// TIA Portal V18 export
TagTable "Screen1_HMI_Tags"
  CV3201_Nuoc_Bon1_M : Real  (PLC tag CV3201_Nuoc_Bon1_M, HMI_Connection_1, 1 s)   // Col1 Bon1, hang CV, PLC_1 addr=%MD1200
  CV3206_Hoi_Bon2_M : Real  (PLC tag CV3206_Hoi_Bon2_M, HMI_Connection_1, 1 s)   // Col2 Bon2, hang CV, PLC_1 addr=%MD1208
  CV3211_Nuoc_Bon3_M : Real  (PLC tag CV3211_Nuoc_Bon3_M, HMI_Connection_2, 1 s)   // Col4 Bon3, hang CV, PLC_2 addr=%MD1216 - BLOCKER
  CV3216_Hoi_Bon4_M : Real  (PLC tag CV3216_Hoi_Bon4_M, HMI_Connection_2, 1 s)   // Col3 Bon4, hang CV, PLC_2 addr=%MD1224 - BLOCKER
  CV3304_Nuoc_Lam_Mat_M : Real  (PLC tag CV3304_Nuoc_Lam_Mat_M, HMI_Connection_1, 1 s)   // x=832,y=741, CV nuoc lam mat, PLC_1 addr=%MD1232, format=999.9 (%)
  FQ3200_Bon1_Eff : Real  (PLC tag FQ3200_Bon1_Eff, HMI_Connection_1, 1 s)   // Col1 Bon1, hang FQ, PLC_1 addr=%MD712
  FQ3205_Bon2_Eff : Real  (PLC tag FQ3205_Bon2_Eff, HMI_Connection_1, 1 s)   // Col2 Bon2, hang FQ, PLC_1 addr=%MD744
  FQ3210_Bon3_Eff : Real  (PLC tag FQ3210_Bon3_Eff, HMI_Connection_2, 1 s)   // Col4 Bon3, hang FQ, PLC_2 addr=%MD776 - BLOCKER
  FQ3215_Bon4_Eff : Real  (PLC tag FQ3215_Bon4_Eff, HMI_Connection_2, 1 s)   // Col3 Bon4, hang FQ, PLC_2 addr=%MD808 - BLOCKER: can HMI_Connection_2
  FT3309_Xa_Thanh_Pham_Eff : Real  (PLC tag FT3309_Xa_Thanh_Pham_Eff, HMI_Connection_1, 1 s)   // x=1280,y=670, FT xa thanh pham, PLC_1 addr=%MD880, format=999.9 (L/h)
  HMI_Anim_Bon1_Frame : Int  (PLC tag HMI_Anim_Bon1_Frame, HMI_Connection_1, 1 s)   // Graphic IOField Graphic I/O field_38 for HMI_Anim_Bon1_Frame
  HMI_Anim_Bon1_MucDich : Int  (PLC tag HMI_Anim_Bon1_MucDich, HMI_Connection_1, 1 s)   // Graphic IOField Graphic I/O field_10 for HMI_Anim_Bon1_MucDich
  HMI_Anim_Bon2_Frame : Int  (PLC tag HMI_Anim_Bon2_Frame, HMI_Connection_1, 1 s)   // Graphic IOField Graphic I/O field_39 for HMI_Anim_Bon2_Frame
  HMI_Anim_Bon2_MucDich : Int  (PLC tag HMI_Anim_Bon2_MucDich, HMI_Connection_1, 1 s)   // Graphic IOField Graphic I/O field_3 for HMI_Anim_Bon2_MucDich
  HMI_Anim_Bon3_Frame : Int  (PLC tag HMI_Anim_Bon3_Frame, HMI_Connection_2, 1 s)   // Graphic IOField Graphic I/O field_41 for HMI_Anim_Bon3_Frame
  HMI_Anim_Bon3_MucDich : Int  (PLC tag HMI_Anim_Bon3_MucDich, HMI_Connection_2, 1 s)   // Graphic IOField Graphic I/O field_6 for HMI_Anim_Bon3_MucDich
  HMI_Anim_Bon4_Frame : Int  (PLC tag HMI_Anim_Bon4_Frame, HMI_Connection_2, 1 s)   // Graphic IOField Graphic I/O field_40 for HMI_Anim_Bon4_Frame
  HMI_Anim_Bon4_MucDich : Int  (PLC tag HMI_Anim_Bon4_MucDich, HMI_Connection_2, 1 s)   // Graphic IOField Graphic I/O field_4 for HMI_Anim_Bon4_MucDich
  HMI_Anim_BonChua1_MucDich : Int  (PLC tag HMI_Anim_BonChua1_MucDich, HMI_Connection_1, 1 s)   // Graphic IOField Graphic I/O field_9 for HMI_Anim_BonChua1_MucDich
  HMI_Anim_BonChua2_MucDich : Int  (PLC tag HMI_Anim_BonChua2_MucDich, HMI_Connection_1, 1 s)   // Graphic IOField Graphic I/O field_2 for HMI_Anim_BonChua2_MucDich
  LT3203_Bon1_Eff : Real  (PLC tag LT3203_Bon1_Eff, HMI_Connection_1, 1 s)   // Col1 Bon1, hang LT, PLC_1 addr=%MD720
  LT3209_Bon2_Eff : Real  (PLC tag LT3209_Bon2_Eff, HMI_Connection_1, 1 s)   // Col2 Bon2, hang LT, PLC_1 addr=%MD752
  LT3213_Bon3_Eff : Real  (PLC tag LT3213_Bon3_Eff, HMI_Connection_2, 1 s)   // Col4 Bon3, hang LT, PLC_2 addr=%MD784 - BLOCKER
  LT3218_Bon4_Eff : Real  (PLC tag LT3218_Bon4_Eff, HMI_Connection_2, 1 s)   // Col3 Bon4, hang LT, PLC_2 addr=%MD816 - BLOCKER
  LT3302_BonChua1_Eff : Real  (PLC tag LT3302_BonChua1_Eff, HMI_Connection_1, 1 s)   // BonChua1 trai, LT muc long, PLC_1 addr=%MD832
  LT3307_BonChua2_Eff : Real  (PLC tag LT3307_BonChua2_Eff, HMI_Connection_1, 1 s)   // BonChua2 phai, LT muc long, PLC_1 addr=%MD856
  PI3308_Truoc_Filter_Eff : Real  (PLC tag PI3308_Truoc_Filter_Eff, HMI_Connection_1, 1 s)   // x=1280,y=616, ap suat truoc filter, PLC_1, format=99.9 (bar)
  Pump3264_Chuyen_Nhanh1 : Bool  (PLC tag Pump3264_Chuyen_Nhanh1, HMI_Connection_1, 1 s)   // Graphic IOField Graphic I/O field_33 for Pump3264_Chuyen_Nhanh1
  Pump3265_Chuyen_Nhanh2 : Bool  (PLC tag Pump3265_Chuyen_Nhanh2, HMI_Connection_2, 1 s)   // Graphic IOField Graphic I/O field_37 for Pump3265_Chuyen_Nhanh2
  Pump3361_LuanChuyen_BonChua1 : Bool  (PLC tag Pump3361_LuanChuyen_BonChua1, HMI_Connection_1, 1 s)   // Graphic IOField Graphic I/O field_34 for Pump3361_LuanChuyen_BonChua1
  Pump3362_Xa_BonChua1 : Bool  (PLC tag Pump3362_Xa_BonChua1, HMI_Connection_1, 1 s)   // Graphic IOField Graphic I/O field_1 for Pump3362_Xa_BonChua1
  Pump3364_Filter : Bool  (PLC tag Pump3364_Filter, HMI_Connection_1, 1 s)   // Graphic IOField Graphic I/O field_35 for Pump3364_Filter
  Pump3365_Filter : Bool  (PLC tag Pump3365_Filter, HMI_Connection_1, 1 s)   // Graphic IOField Graphic I/O field_36 for Pump3365_Filter
  TT3204_Bon1_Eff : Real  (PLC tag TT3204_Bon1_Eff, HMI_Connection_1, 1 s)   // Col1 Bon1, hang TT, PLC_1 addr=%MD728
  TT3208_Bon2_Eff : Real  (PLC tag TT3208_Bon2_Eff, HMI_Connection_1, 1 s)   // Col2 Bon2, hang TT, PLC_1 addr=%MD760
  TT3214_Bon3_Eff : Real  (PLC tag TT3214_Bon3_Eff, HMI_Connection_2, 1 s)   // Col4 Bon3, hang TT, PLC_2 addr=%MD792 - BLOCKER
  TT3219_Bon4_Eff : Real  (PLC tag TT3219_Bon4_Eff, HMI_Connection_2, 1 s)   // Col3 Bon4, hang TT, PLC_2 addr=%MD824 - BLOCKER
  TT3301_BonChua1_Eff : Real  (PLC tag TT3301_BonChua1_Eff, HMI_Connection_1, 1 s)   // BonChua1 trai, TT nhiet do, PLC_1 addr=%MD840
  TT3303_TraoDoiNhiet_Eff : Real  (PLC tag TT3303_TraoDoiNhiet_Eff, HMI_Connection_1, 1 s)   // x=791,y=589, TT trao doi nhiet, PLC_1 addr=%MD848, format=99.9 (°C)
  TT3306_BonChua2_Eff : Real  (PLC tag TT3306_BonChua2_Eff, HMI_Connection_1, 1 s)   // BonChua2 phai, TT nhiet do, PLC_1 addr=%MD864
  V3230_Nuoc_Bon1 : Bool  (PLC tag V3230_Nuoc_Bon1, HMI_Connection_1, 1 s)   // Graphic IOField Graphic I/O field_5 for V3230_Nuoc_Bon1
  V3232_Xa_Bon1 : Bool  (PLC tag V3232_Xa_Bon1, HMI_Connection_1, 1 s)   // Graphic IOField Graphic I/O field_8 for V3232_Xa_Bon1
  V3233_Xa_Bon1 : Bool  (PLC tag V3233_Xa_Bon1, HMI_Connection_1, 1 s)   // Graphic IOField Graphic I/O field_7 for V3233_Xa_Bon1
  V3234_Xa_Bon1 : Bool  (PLC tag V3234_Xa_Bon1, HMI_Connection_1, 1 s)   // Graphic IOField Graphic I/O field_11 for V3234_Xa_Bon1
  V3235_Nuoc_Bon2 : Bool  (PLC tag V3235_Nuoc_Bon2, HMI_Connection_1, 1 s)   // Graphic IOField Graphic I/O field_12 for V3235_Nuoc_Bon2
  V3237_Xa_Bon2 : Bool  (PLC tag V3237_Xa_Bon2, HMI_Connection_1, 1 s)   // Graphic IOField Graphic I/O field_15 for V3237_Xa_Bon2
  V3238_Xa_Bon2 : Bool  (PLC tag V3238_Xa_Bon2, HMI_Connection_1, 1 s)   // Graphic IOField Graphic I/O field_17 for V3238_Xa_Bon2
  V3239_Xa_Bon2 : Bool  (PLC tag V3239_Xa_Bon2, HMI_Connection_1, 1 s)   // Graphic IOField Graphic I/O field_16 for V3239_Xa_Bon2
  V3240_Nuoc_Bon3 : Bool  (PLC tag V3240_Nuoc_Bon3, HMI_Connection_2, 1 s)   // Graphic IOField Graphic I/O field_14 for V3240_Nuoc_Bon3
  V3242_Xa_Bon3 : Bool  (PLC tag V3242_Xa_Bon3, HMI_Connection_2, 1 s)   // Graphic IOField Graphic I/O field_19 for V3242_Xa_Bon3
  V3243_Xa_Bon3 : Bool  (PLC tag V3243_Xa_Bon3, HMI_Connection_2, 1 s)   // Graphic IOField Graphic I/O field_23 for V3243_Xa_Bon3
  V3244_Xa_Bon3 : Bool  (PLC tag V3244_Xa_Bon3, HMI_Connection_2, 1 s)   // Graphic IOField Graphic I/O field_21 for V3244_Xa_Bon3
  V3245_Nuoc_Bon4 : Bool  (PLC tag V3245_Nuoc_Bon4, HMI_Connection_2, 1 s)   // Graphic IOField Graphic I/O field_13 for V3245_Nuoc_Bon4
  V3247_Xa_Bon4 : Bool  (PLC tag V3247_Xa_Bon4, HMI_Connection_2, 1 s)   // Graphic IOField Graphic I/O field_18 for V3247_Xa_Bon4
  V3248_Xa_Bon4 : Bool  (PLC tag V3248_Xa_Bon4, HMI_Connection_2, 1 s)   // Graphic IOField Graphic I/O field_22 for V3248_Xa_Bon4
  V3249_Xa_Bon4 : Bool  (PLC tag V3249_Xa_Bon4, HMI_Connection_2, 1 s)   // Graphic IOField Graphic I/O field_20 for V3249_Xa_Bon4
  V3331_Xa_BonChua1 : Bool  (PLC tag V3331_Xa_BonChua1, HMI_Connection_1, 1 s)   // Graphic IOField Graphic I/O field_24 for V3331_Xa_BonChua1
  V3332_Xa_BonChua1 : Bool  (PLC tag V3332_Xa_BonChua1, HMI_Connection_1, 1 s)   // Graphic IOField Graphic I/O field_30 for V3332_Xa_BonChua1
  V3333_DieuHuong_BonChua1 : Bool  (PLC tag V3333_DieuHuong_BonChua1, HMI_Connection_1, 1 s)   // Graphic IOField Graphic I/O field_27 for V3333_DieuHuong_BonChua1
  V3334_DieuHuong_BonChua1 : Bool  (PLC tag V3334_DieuHuong_BonChua1, HMI_Connection_1, 1 s)   // Graphic IOField Graphic I/O field_25 for V3334_DieuHuong_BonChua1
  V3335_DieuHuong_BonChua1 : Bool  (PLC tag V3335_DieuHuong_BonChua1, HMI_Connection_1, 1 s)   // Graphic IOField Graphic I/O field_26 for V3335_DieuHuong_BonChua1
  V3338_Xa_BonChua2 : Bool  (PLC tag V3338_Xa_BonChua2, HMI_Connection_1, 1 s)   // Graphic IOField Graphic I/O field_28 for V3338_Xa_BonChua2
  V3339_Xa_BonChua2 : Bool  (PLC tag V3339_Xa_BonChua2, HMI_Connection_1, 1 s)   // Graphic IOField Graphic I/O field_31 for V3339_Xa_BonChua2
  V3340_Duong_Filter : Bool  (PLC tag V3340_Duong_Filter, HMI_Connection_1, 1 s)   // Graphic IOField Graphic I/O field_32 for V3340_Duong_Filter
  V3341_Duong_Filter : Bool  (PLC tag V3341_Duong_Filter, HMI_Connection_1, 1 s)   // Graphic IOField Graphic I/O field_29 for V3341_Duong_Filter
  GIA_TRI_NHIET_DO_DOC_VE : Real  (1 s)   // Dummy internal tag for bon tron 1 temperature
  nguyen_lieu_tron_1 : Bool  (1 s)   // Dummy internal tag for bon tron 1 material
  cap_nuoc_tron_1 : Bool  (1 s)   // Dummy internal tag for bon tron 1 water
  start : Bool  (1 s)   // Dummy internal tag for bon tron 1 start button
  HMI_SP_PLC1_Nuoc_Bon1 : Real  (PLC tag HMI_SP_PLC1_Nuoc_Bon1, HMI_Connection_1, 1 s)
  HMI_SP_PLC1_Nuoc_Bon2 : Real  (PLC tag HMI_SP_PLC1_Nuoc_Bon2, HMI_Connection_1, 1 s)
  HMI_SP_PLC1_Nhiet_Do_Bon2 : Real  (PLC tag HMI_SP_PLC1_Nhiet_Do_Bon2, HMI_Connection_1, 1 s)
  HMI_SP_PLC2_Nuoc_Bon3 : Real  (PLC tag HMI_SP_PLC2_Nuoc_Bon3, HMI_Connection_2, 1 s)
  HMI_SP_PLC2_Nuoc_Bon4 : Real  (PLC tag HMI_SP_PLC2_Nuoc_Bon4, HMI_Connection_2, 1 s)
  HMI_SP_PLC2_Nhiet_Do_Bon4 : Real  (PLC tag HMI_SP_PLC2_Nhiet_Do_Bon4, HMI_Connection_2, 1 s)
  HMI_SP_Time_Khuay_Bon1 : Time  (PLC tag HMI_SP_Time_Khuay_Bon1, HMI_Connection_1, 1 s)
  HMI_SP_Time_Khuay_Bon3 : Time  (PLC tag HMI_SP_Time_Khuay_Bon3, HMI_Connection_2, 1 s)
  HMI_SP_Time_Fwd : Time  (PLC tag HMI_SP_Time_Fwd, HMI_Connection_1, 1 s)
  HMI_SP_Time_Rev : Time  (PLC tag HMI_SP_Time_Rev, HMI_Connection_1, 1 s)
  HMI_SP_Time_Sterilize : Time  (PLC tag HMI_SP_Time_Sterilize, HMI_Connection_1, 1 s)
